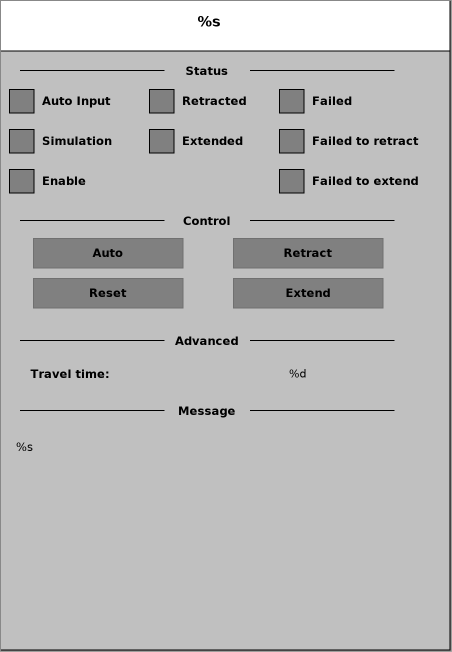
VISUALIZATION Cylinder_Template  // 452x652
VAR_IN_OUT
	DUT										: DUT_Cylinder;
END_VAR
    Group (0,0 418x530)
        Rectangle (0,0 450x650)
        Rectangle (0,0 450x51)
    Label (132,56 150x30), "Status"
    Line (20,70) (164,70)
    Label (132,206 150x30), "Control"
    Label (132,326 150x30), "Advanced"
    Label (132,396 150x30), "Message"
    Textfield (0,3 418x37), "%s", text variable: DUT.CylinderID
    RoundedRectangle (9,89 25x24), colour toggle: DUT.AutInp
    Label (39,86 106x30), "Auto Input"
    Label (39,126 106x30), "Simulation"
    RoundedRectangle (9,129 25x24), colour toggle: DUT.Simulate
    Label (39,166 106x30), "Enable"
    RoundedRectangle (9,169 25x24), colour toggle: DUT.Enable
    RoundedRectangle (279,89 25x24), colour toggle: DUT.Failed
    Label (309,86 106x30), "Failed"
    Label (309,126 106x30), "Failed to retract"
    RoundedRectangle (279,129 25x24), colour toggle: DUT.Failed_To_Retract
    Label (309,166 106x30), "Failed to extend"
    RoundedRectangle (279,169 25x24), colour toggle: DUT.Failed_To_Extend
    Button (33,238 150x30), "Auto", colour toggle: DUT.CMD = 4
        OnMouseClick: execute { DUT.CMD			:= 4; }
    Button (33,278 150x30), "Reset", colour toggle: DUT.Reset
        toggle DUT.Reset
    Button (233,238 150x30), "Retract", colour toggle: DUT.CMD = 1
        OnMouseClick: execute { DUT.CMD			:= 1; }
    Button (233,278 150x30), "Extend", colour toggle: DUT.CMD = 2
        OnMouseClick: execute { DUT.CMD			:= 2; }
    Label (16,359 108x30), "Travel time:"
    Textfield (223,359 150x30), "%d", text variable: DUT.Travel_Time
        OnMouseClick: write DUT.Travel_Time via Default, min 1, max 999
    Textfield (13,439 392x76), "%s", text variable: DUT.Message
    Line (250,70) (394,70)
    Line (250,220) (394,220)
    Line (20,220) (164,220)
    Line (250,340) (394,340)
    Line (20,340) (164,340)
    Line (250,410) (394,410)
    Line (20,410) (164,410)
    RoundedRectangle (149,89 25x24), colour toggle: DUT.Retracted
    Label (179,86 106x30), "Retracted"
    Label (179,126 106x30), "Extended"
    RoundedRectangle (149,129 25x24), colour toggle: DUT.Extended
END_VISUALIZATION

(* stored: Version 1.1.0.1, ProductVersion 3.1.4022.18
   Visu Cylinder_Template: Id {f8c447f8-da2e-4c40-86fa-d4198f22ef1e} *)
